FUNCTION_BLOCK FB_SendDriveReset
VAR_INPUT
	DriveReset : INT;
END_VAR
VAR_OUTPUT
END_VAR
VAR
	TxMessage : EXTCANQUEUE;
END_VAR
VAR_IN_OUT
	CAN_OUTPUTS : CANTXQUEUESTRUCT_E_32;
	CAN_INPUTS : CANRXQUEUESTRUCT_E_32;
END_VAR

 
TxMessage.cobId := 150;
TxMessage.length := 1;
TxMessage.data[0] :=  INT_TO_BYTE(DriveReset AND 16#FF);
CAN_OUTPUTS.TxMessages[8] := TxMessage;
//CAN_OUTPUTS.NoOfTxMessages := 1;

(*
TxMessage.cobId := 120;
TxMessage.length := 1;
TxMessage.data[0] :=  INT_TO_BYTE(PropFlag AND 16#FF);
CAN_OUTPUTS.TxMessages[5] := TxMessage;
CAN_OUTPUTS.TxCounter := CAN_INPUTS.TxCounter + 1;
*)

END_FUNCTION_BLOCK

(* stored: Version 1.1.0.1
   POU FB_SendDriveReset: Id {1175849d-ee68-4283-90bd-3fb54b7e7e4a}, SpecialFunc None *)
